FUNCTION_BLOCK FB_RejectCart EXTENDS FB_Machine
VAR_INPUT
	// Device identification
	sLockCylinerID					: STRING;
	
	// Safety box permissive for release and remove cart
	bSafetyBox_permissive			: BOOL;
	
	// Reject request
	bPlacePieceOnCartRequest		: BOOL;
END_VAR
VAR_OUTPUT
	// Safety box enter permissive
	bSafetyBox_okForEnter			: BOOL;
	
	// Request for pieces removal when cart is full
	bRemovePiecesRequest			: BOOL;
	
	// Sensors presence array
	byAvailableNests				: BYTE;
END_VAR
VAR
	// Timmers for considering cart in place
	tonCartIsInPlace				: TON;
	
	// Timmers for considering cart removed
	tonCartRemoved					: TON;

	// Occuped nests in reject cart
	siOccupedNests					: SINT;
	
	// Cart is in position sensor
	bCartPresence					AT %I* : BOOL;
	// 8 sensor array
	byRejectNestsSensors			AT %I* : BYTE;

	// Cylinder for locking the cart in place
	fbCartLock						: FB_Cylinder;
END_VAR

	CountNests();

//	Run the standar main for any machine
	SUPER^.MachineMain();

//	Safety permisive conditions for any device
	fbCartLock(						diStationState:=diStationState,
									sDeviceID:='',
									bStopExecution:=bStopExecution,
									bAlarmReset:=bAlarmReset,
									bPermisiveExtend:= bCartPresence AND bSafetyBox_permissive,
									bPermisiveRetract:= bCartPresence AND bSafetyBox_permissive,
									Timeout:= T#1S);
	fbCartLock.bExtendRequest		:=FALSE;
	fbCartLock.bRetractRequest		:=FALSE;

METHOD  Alarm
//	Step timeout
	ton_StepTimeout(					IN:= diActualSeqStep=diLastActiveStep,
										PT:= T#1S);

// 	Following of sequence for setting timeout
	IF diLastActiveStep<>diActualSeqStep THEN
		diLastActiveStep					:= diActualSeqStep;
	END_IF

//	For setting an sequence alarm code
	IF ton_StepTimeout.Q THEN
		CASE diActualSeqStep OF
			10: 	sAlarm				:= '';	// Init wait cart in position timeout
			50: 	sAlarm				:= '';	// Cart clamping timeout
			110: 	sAlarm				:= '';	// Cart removal timeout
			1000: 	sAlarm				:= '';	// Cart in position and clamped timeout
			1100: 	sAlarm				:= '';	// Cart removal timeout
		END_CASE
	END_IF

//	Concat general alarm codes with cart lock cylinder alarm codes
	sAlarm								:= CONCAT(STR1:=sAlarm,STR2:=fbCartLock.sAlarm);
END_METHOD

METHOD  Auto
//	Keep sequencer in range
	IF diActualSeqStep<1000 OR diActualSeqStep>1999 THEN
		diActualSeqStep					:= 1000;
	END_IF

CASE diActualSeqStep OF
	1000:								//	Check for cart in position and it is clamped
		IF tonCartIsInPlace.Q AND fbCartLock.bIsExtended THEN
			fbCartLock.bRetractRequest	:= FALSE;
			fbCartLock.bExtendRequest	:= FALSE;
			diActualSeqStep				:= 1050;
	
		ELSIF tonCartIsInPlace.Q AND fbCartLock.bIsRetracted THEN
			fbCartLock.bRetractRequest	:= FALSE;
			fbCartLock.bExtendRequest	:= TRUE;
	
		ELSE
			fbCartLock.bExtendRequest	:= FALSE;
			fbCartLock.bRetractRequest	:= TRUE;
		END_IF
	1050:								//	If there are not availability of places in cart release it and wait it has been removed
		IF siOccupedNests>=8 THEN
			fbCartLock.bExtendRequest	:= FALSE;
			fbCartLock.bRetractRequest	:= TRUE;
		END_IF
		IF fbCartLock.bIsRetracted THEN
			diActualSeqStep				:= 1100;
		END_IF
	1100:								//	Waiting cart removal
		IF tonCartRemoved.Q THEN
			diActualSeqStep				:= 1000;
		END_IF
END_CASE
END_METHOD

ACTION CountNests:
//  Counts occuped nests in the cart
	siOccupedNests					:= 0;
	IF byRejectNestsSensors.0 THEN
		siOccupedNests				:= siOccupedNests + 1;
	END_IF
	IF byRejectNestsSensors.1 THEN
		siOccupedNests				:= siOccupedNests + 1;
	END_IF
	IF byRejectNestsSensors.2 THEN
		siOccupedNests				:= siOccupedNests + 1;
	END_IF
	IF byRejectNestsSensors.3 THEN
		siOccupedNests				:= siOccupedNests + 1;
	END_IF
	IF byRejectNestsSensors.4 THEN
		siOccupedNests				:= siOccupedNests + 1;
	END_IF
	IF byRejectNestsSensors.5 THEN
		siOccupedNests				:= siOccupedNests + 1;
	END_IF
	IF byRejectNestsSensors.6 THEN
		siOccupedNests				:= siOccupedNests + 1;
	END_IF
	IF byRejectNestsSensors.7 THEN
		siOccupedNests				:= siOccupedNests + 1;
	END_IF
END_ACTION

METHOD  Init
//	Keep sequencer in range
	IF diActualSeqStep<0 OR diActualSeqStep>999 THEN
		diActualSeqStep					:= 0;
	END_IF

CASE diActualSeqStep OF
	0:									//	Wait for the initial permisive and reset values
		IF  bInit_StartPermissive THEN
			fbCartLock.bRetractRequest	:= FALSE;
			fbCartLock.bExtendRequest	:= FALSE;
			diActualSeqStep 			:= 10;
		END_IF
	10:									// Check cart is in place
		IF tonCartIsInPlace.Q THEN
			diActualSeqStep 			:= 50;
		ELSE
			fbCartLock.bRetractRequest:=TRUE;
		END_IF
	50:									// Confirm cart is clamped
		fbCartLock.bRetractRequest		:= FALSE;
		fbCartLock.bExtendRequest		:= TRUE;
		IF fbCartLock.bIsExtended THEN
			fbCartLock.bExtendRequest	:= FALSE;
			diActualSeqStep				:= 100;
		END_IF
	100:								// Check reject nest availability for release cart
		IF siOccupedNests>=4 THEN
			diActualSeqStep				:= 110;
		ELSE
			diActualSeqStep 			:= 999;
		END_IF
	110:								// Unlock cart and wait it's removed
		bRemovePiecesRequest			:= TRUE;
		fbCartLock.bRetractRequest		:= TRUE;
		IF fbCartLock.bIsRetracted AND tonCartRemoved.Q THEN
			diActualSeqStep				:= 0;
		END_IF
	999:								// Init finished
		bInit_Finished					:= TRUE;
END_CASE
END_METHOD

METHOD  IO
//	For considering cart in place
	tonCartIsInPlace(							IN:=bCartPresence,
												PT:=T#1S);

//	For considering cart has been removed
	tonCartRemoved(							IN:=NOT bCartPresence,
												PT:=T#1S);

//	If all places are ocupped request cart removal
	IF siOccupedNests>=8 THEN
		bRemovePiecesRequest				:= TRUE;
//	If cart is removed clear request
	ELSIF tonCartRemoved.Q THEN
		bRemovePiecesRequest				:= FALSE;
	END_IF

//	Piece sensor inverse polaritiy refreshing in available positions var
	IF tonCartIsInPlace.Q AND fbCartLock.bIsExtended THEN
		byAvailableNests.0						:= NOT byRejectNestsSensors.0;
		byAvailableNests.1						:= NOT byRejectNestsSensors.1;
		byAvailableNests.2						:= NOT byRejectNestsSensors.2;
		byAvailableNests.3						:= NOT byRejectNestsSensors.3;
		byAvailableNests.4						:= NOT byRejectNestsSensors.4;
		byAvailableNests.5						:= NOT byRejectNestsSensors.5;
		byAvailableNests.6						:= NOT byRejectNestsSensors.6;
		byAvailableNests.7						:= NOT byRejectNestsSensors.7;
	ELSE
		byAvailableNests						:= 0;
	END_IF

//	For safety box enter permissive
	bSafetyBox_okForEnter						:= tonCartIsInPlace.Q AND fbCartLock.bIsExtended;
END_METHOD

METHOD  Manual
END_METHOD

METHOD  Pause
END_METHOD

METHOD  Stop
END_METHOD

END_FUNCTION_BLOCK

(* stored: Version 1.1.0.1, ProductVersion 3.1.4024.12
   POU FB_RejectCart: Id {743a376f-4fa0-4fba-821c-e0b7d34bd821}, SpecialFunc None
   Method Alarm: Id {a2e3233f-e38e-4263-92eb-523118066f8e}
   Method Auto: Id {ceee8003-41cf-4c72-a85c-d9e2b0f68d8c}
   Action CountNests: Id {3b2313c9-83b0-41af-9e3b-f1539f266f22}
   Method Init: Id {fcbb3f26-0058-4481-9c58-3d096317d08f}
   Method IO: Id {39def025-d6fb-42e4-a8f1-838c4d1768f8}
   Method Manual: Id {bd5d7f9f-2e54-42b2-b27b-2eaea211983d}
   Method Pause: Id {1af13883-64d8-4728-bf6f-b440c3dfa3ac}
   Method Stop: Id {84642c77-2ff7-4ecd-b4e9-c68a1daa0f7e} *)
